// TIA Portal V20 export
DATA_BLOCK "PM02"   // DB336
// stored: MemoryReserve 100
   VAR
      "SUCTION PAD #1 TOP UP" : Bool := FALSE;
      "SUCTION PAD #1 TOP DOWN" : Bool := FALSE;
      "SUCTION PAD #1 BTM UP" : Bool := FALSE;
      "SUCTION PAD #1 BTM DOWN" : Bool := FALSE;
      "CUTTER #1 UP" : Bool := FALSE;
      "CUTTER #1 DOWN" : Bool := FALSE;
      "TAPE #1 TOP UP" : Bool := FALSE;
      "TAPE #1 TOP DOWN" : Bool := FALSE;
      "TAPE #1 BTM UP" : Bool := FALSE;
      "TAPE #1 BTM DOWN" : Bool := FALSE;
      "SPLICE HEAD ROTATE #1 TOP FORWARD" : Bool := FALSE;
      "SPLICE HEAD ROTATE #1 TOP BACKWARD" : Bool := FALSE;
      "SPLICE HEAD ROTATE #1 BTM FORWARD" : Bool := FALSE;
      "SPLICE HEAD ROTATE #1 BTM BACKWARD" : Bool := FALSE;
   END_VAR
BEGIN
END_DATA_BLOCK
